(* PLC project rootsystem, Dassault Systèmes ControlBuild 2024x Refresh1 *)
(* stored: creationDateTime 2024-03-13T17:20:51-01:00 *)

PROGRAM mac
  VAR_IN_OUT
    con : REAL := 0.0;
  END_VAR

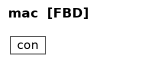
(* FBD diagram, written out as Structured Text *)
END_PROGRAM

PROGRAM my_app.rootsystem
  VAR_INPUT
    aaaaa : REAL := 0.0;
  END_VAR
  VAR_OUTPUT
    bbbb : REAL := 0.0;
  END_VAR

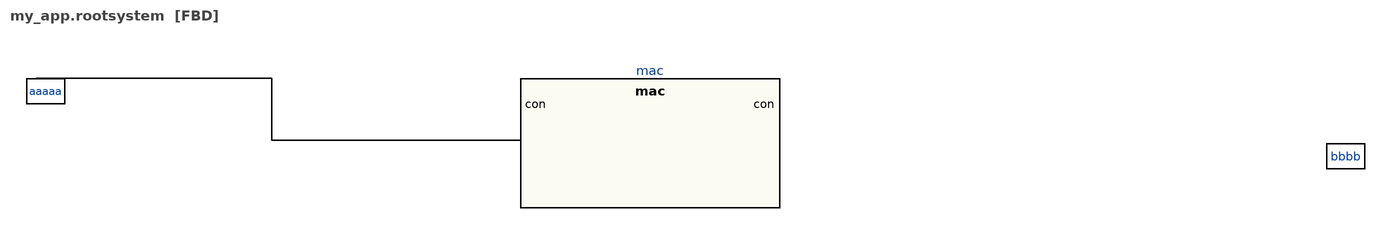
(* FBD diagram, written out as Structured Text *)
mac(con := aaaaa);
END_PROGRAM
